(* LS Electric XG5000 project: elevator *)
(* PLC LSPLC *)
(* module base 0 slot 0: FEnet:XGL-EFMT(B) (Fast Ethernet 통신 모듈, 전기 Master) *)
(* module base 0 slot 1: 입력 모듈:XGI-D21A (DC 24V 입력, 8점 (전류소스/싱크입력)) *)
(* module base 0 slot 2: 출력 모듈:XGQ-RY1A (릴레이 출력, 8점 (2A용, 단독 COM.)) *)

(* Comments on direct variables
%IX0.1.0	1층 외부 ▲
%IX0.1.1	2층 외부  ▲
%IX0.1.2	2층 외부 ▼
%IX0.1.3	3층 외부  ▲
%IX0.1.4	3층 외부 ▼
%IX0.1.5	4층 외부  ▲
%IX0.1.6	4층 외부 ▼
%IX0.1.7	5층 외부 ▼
%IX0.3.0	내부 목적지 1F
%IX0.3.1	내부 목적지 2F
%IX0.3.2	내부 목적지 3F
%IX0.3.3	내부 목적지 4F
%IX0.3.4	내부 목적지 5F
%IX0.3.5	문 열기
%IX0.3.6	문 닫기
%IX0.3.7	비상정지
%MX80	1층 상승
%MX81	2층 상승
%MX82	3층 상승
%MX83	4층 상승
%MX89	2층 하강
%MX90	3층 하강
%MX91	4층 하강
%MX92	5층 하강
%MX96	1층
%MX97	2층
%MX98	3층
%MX99	4층
%MX100	5층
%MX160	비상정지
%MX161	문 닫힘 / 이동 가능
%MX162	문 열리는 중
%MX163	문 완전 열림
%MX164	문 딛히는 중
%MX165	상승 가능
%MX166	하강 가능
%MX167	초기화용
%MX176	1층 호출 있음
%MX177	2층 호출 있음
%MX178	3층 호출 있음
%MX179	4층 호출 있음
%MX180	5층 호출 있음
%MX181	내부 큐 있음
%MX240	외부 입력 1▲
%MX241	외부 입력 2▲
%MX242	외부 입력 2▼
%MX243	외부 입력 3▲
%MX244	외부 입력 3▼
%MX245	외부 입력 4▲
%MX246	외부 입력 4▼
%MX247	외부 입력 5▼
%MX248	내부 입력 1F
%MX249	내부 입력 2F
%MX250	내부 입력 3F
%MX251	내부 입력 4F
%MX252	내부 입력 5F
%MX253	내부입력 문열기
%MX254	내부입력 문닫기
%MX255	내부 비상정지
%MB10	상승 큐
%MB11	하강 큐
%MB12	내부 큐
%MW0	현재 층
%MW1	목표 층
%MW2	이동 방향
%MW3	상태
%MW4	TO.ET 전달용
%QX0.4.0	1층 표시등
%QX0.4.1	2층 표시등
%QX0.4.2	3층 표시등
%QX0.4.3	4층 표시등
%QX0.4.4	5층 표시등
%QX0.4.5	상승 ▲ 표시등
%QX0.4.6	하강 ▼ 표시등
%QX0.4.7	비상정지 표시등
*)

PROGRAM 리셋 (* task: 스캔 프로그램 *)
VAR
    _p1 : BOOL;
END_VAR

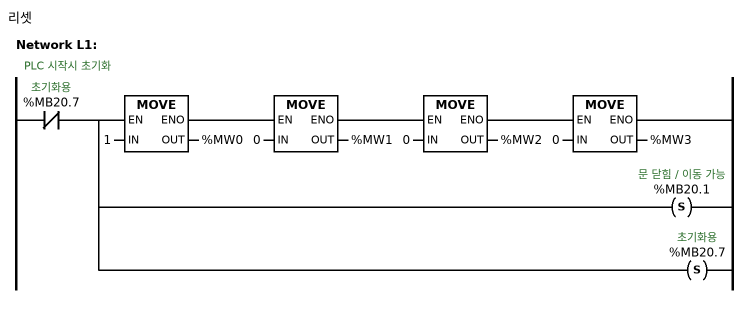
(* PLC 시작시 초기화 *)
(* Rung L1 *)
IF NOT %MB20.7 THEN
    %MW0 := 1;
    %MW1 := 0;
    %MW2 := 0;
    %MW3 := 0;
END_IF;
_p1 := NOT %MB20.7;
IF _p1 THEN
    %MB20.1 := TRUE;
    %MB20.7 := TRUE;
END_IF;
END_PROGRAM

PROGRAM 비상정지 (* task: 스캔 프로그램 *)
VAR
    _p1 : BOOL;
    _p2 : BOOL;
END_VAR

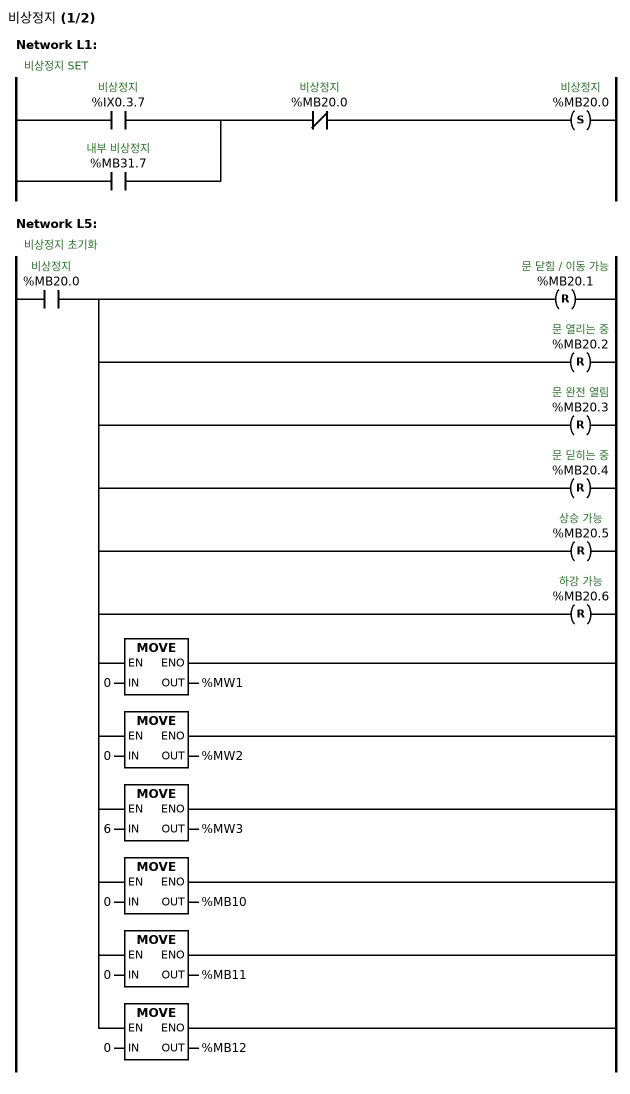
(* 비상정지 SET *)
(* Rung L1 *)
IF (%IX0.3.7 OR %MB31.7) AND NOT %MB20.0 THEN %MB20.0 := TRUE; END_IF;
(* 비상정지 초기화 *)
(* Rung L5 *)
_p1 := %MB20.0;
IF _p1 THEN
    %MB20.1 := FALSE;
    %MB20.2 := FALSE;
    %MB20.3 := FALSE;
    %MB20.4 := FALSE;
    %MB20.5 := FALSE;
    %MB20.6 := FALSE;
    %MW1 := 0;
    %MW2 := 0;
    %MW3 := 6;
    %MB10 := 0;
    %MB11 := 0;
    %MB12 := 0;
END_IF;

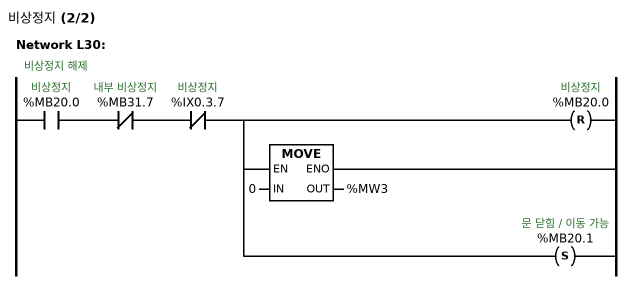
(* 비상정지 해제 *)
(* Rung L30 *)
_p2 := %MB20.0 AND NOT %MB31.7 AND NOT %IX0.3.7;
IF _p2 THEN
    %MB20.0 := FALSE;
    %MW3 := 0;
    %MB20.1 := TRUE;
END_IF;
END_PROGRAM

PROGRAM 호출큐등록 (* task: 스캔 프로그램 *)

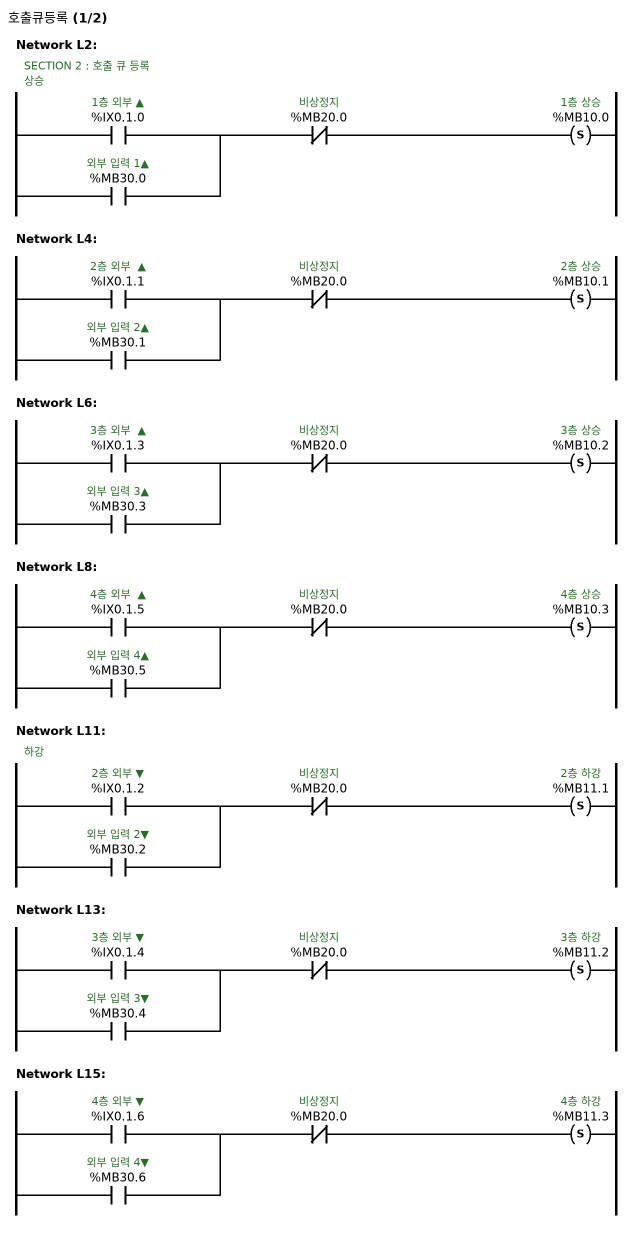
(* SECTION 2 : 호출 큐 등록 *)
(* 상승 *)
(* Rung L2 *)
IF (%IX0.1.0 OR %MB30.0) AND NOT %MB20.0 THEN %MB10.0 := TRUE; END_IF;
(* Rung L4 *)
IF (%IX0.1.1 OR %MB30.1) AND NOT %MB20.0 THEN %MB10.1 := TRUE; END_IF;
(* Rung L6 *)
IF (%IX0.1.3 OR %MB30.3) AND NOT %MB20.0 THEN %MB10.2 := TRUE; END_IF;
(* Rung L8 *)
IF (%IX0.1.5 OR %MB30.5) AND NOT %MB20.0 THEN %MB10.3 := TRUE; END_IF;
(* 하강 *)
(* Rung L11 *)
IF (%IX0.1.2 OR %MB30.2) AND NOT %MB20.0 THEN %MB11.1 := TRUE; END_IF;
(* Rung L13 *)
IF (%IX0.1.4 OR %MB30.4) AND NOT %MB20.0 THEN %MB11.2 := TRUE; END_IF;
(* Rung L15 *)
IF (%IX0.1.6 OR %MB30.6) AND NOT %MB20.0 THEN %MB11.3 := TRUE; END_IF;

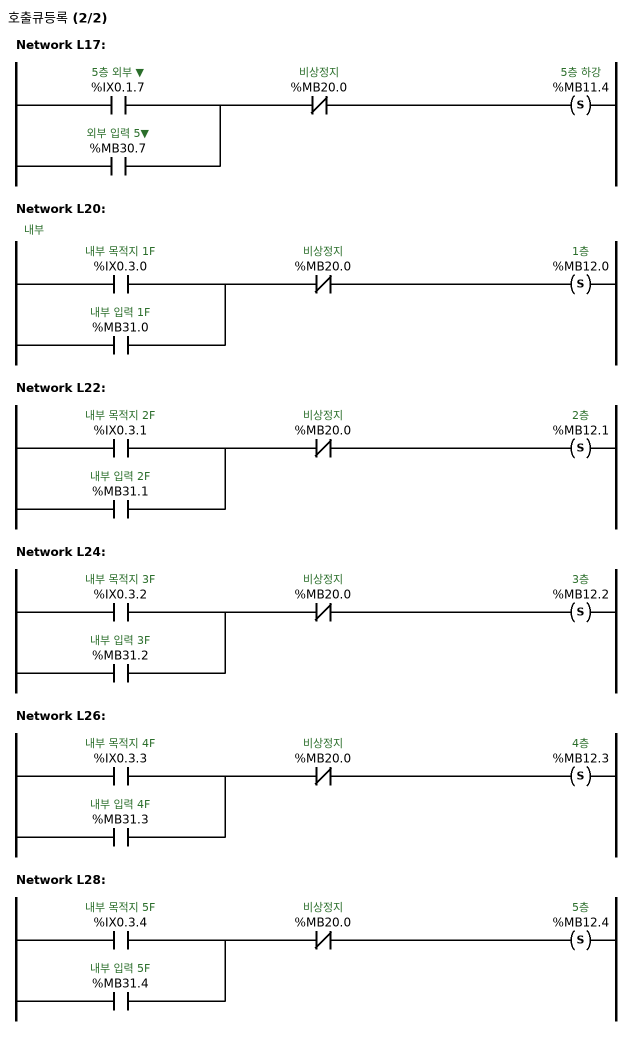
(* Rung L17 *)
IF (%IX0.1.7 OR %MB30.7) AND NOT %MB20.0 THEN %MB11.4 := TRUE; END_IF;
(* 내부 *)
(* Rung L20 *)
IF (%IX0.3.0 OR %MB31.0) AND NOT %MB20.0 THEN %MB12.0 := TRUE; END_IF;
(* Rung L22 *)
IF (%IX0.3.1 OR %MB31.1) AND NOT %MB20.0 THEN %MB12.1 := TRUE; END_IF;
(* Rung L24 *)
IF (%IX0.3.2 OR %MB31.2) AND NOT %MB20.0 THEN %MB12.2 := TRUE; END_IF;
(* Rung L26 *)
IF (%IX0.3.3 OR %MB31.3) AND NOT %MB20.0 THEN %MB12.3 := TRUE; END_IF;
(* Rung L28 *)
IF (%IX0.3.4 OR %MB31.4) AND NOT %MB20.0 THEN %MB12.4 := TRUE; END_IF;
END_PROGRAM

PROGRAM 방향판별 (* task: 스캔 프로그램 *)
VAR
    _t1 : BOOL;
    _t2 : BOOL;
    _t3 : BOOL;
    _t4 : BOOL;
    _t5 : BOOL;
    _t6 : BOOL;
    _p7 : BOOL;
    _t8 : BOOL;
    _t9 : BOOL;
    _t10 : BOOL;
    _t11 : BOOL;
    _t12 : BOOL;
    _t13 : BOOL;
    _t14 : BOOL;
    _t15 : BOOL;
    _t16 : BOOL;
    _t17 : BOOL;
    _t18 : BOOL;
    _t19 : BOOL;
    _t20 : BOOL;
    _t21 : BOOL;
    _t22 : BOOL;
    _t23 : BOOL;
    _t24 : BOOL;
    _t25 : BOOL;
END_VAR

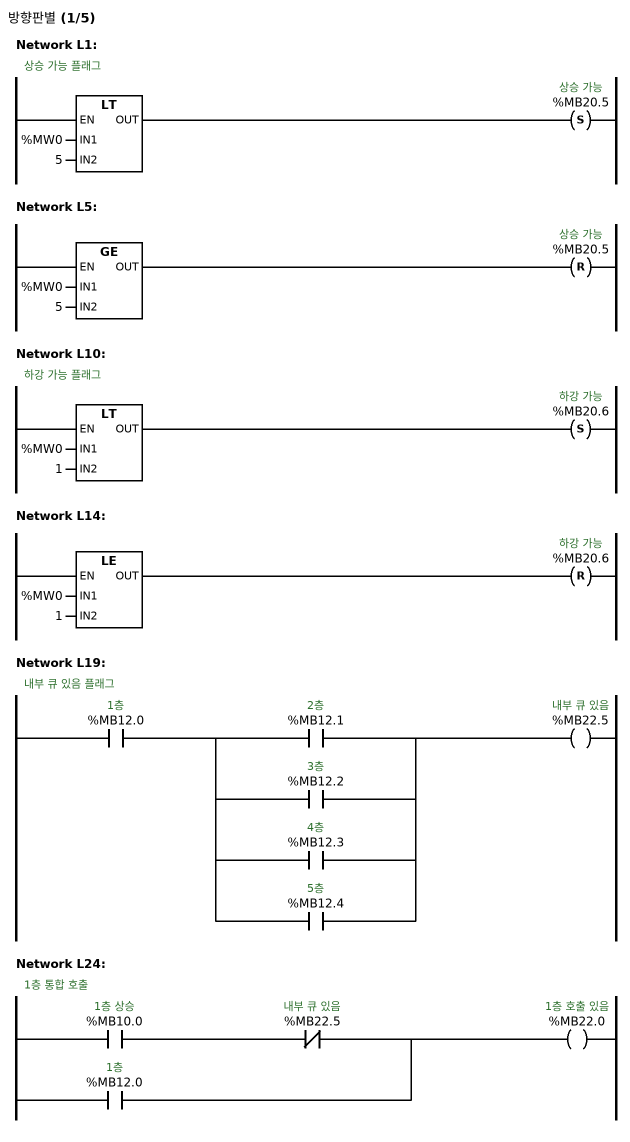
(* 상승 가능 플래그 *)
(* Rung L1 *)
IF %MW0 < 5 THEN %MB20.5 := TRUE; END_IF;
(* Rung L5 *)
IF %MW0 >= 5 THEN %MB20.5 := FALSE; END_IF;
(* 하강 가능 플래그 *)
(* Rung L10 *)
IF %MW0 < 1 THEN %MB20.6 := TRUE; END_IF;
(* Rung L14 *)
IF %MW0 <= 1 THEN %MB20.6 := FALSE; END_IF;
(* 내부 큐 있음 플래그 *)
(* Rung L19 *)
%MB22.5 := %MB12.0 AND (%MB12.1 OR %MB12.2 OR %MB12.3 OR %MB12.4);
(* 1층 통합 호출 *)
(* Rung L24 *)
%MB22.0 := (%MB10.0 AND NOT %MB22.5) OR %MB12.0;

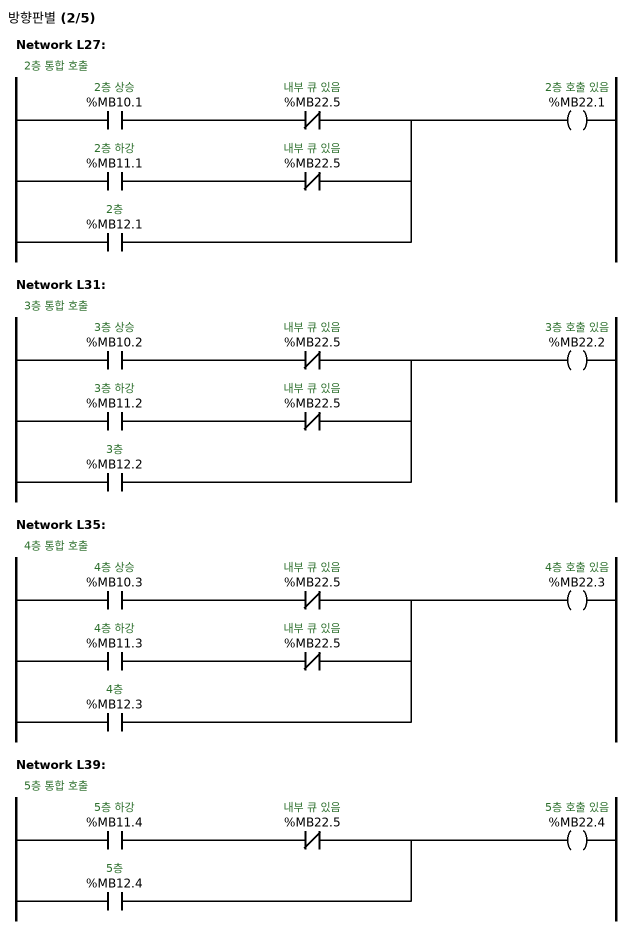
(* 2층 통합 호출 *)
(* Rung L27 *)
%MB22.1 := (%MB10.1 AND NOT %MB22.5) OR (%MB11.1 AND NOT %MB22.5) OR %MB12.1;
(* 3층 통합 호출 *)
(* Rung L31 *)
%MB22.2 := (%MB10.2 AND NOT %MB22.5) OR (%MB11.2 AND NOT %MB22.5) OR %MB12.2;
(* 4층 통합 호출 *)
(* Rung L35 *)
%MB22.3 := (%MB10.3 AND NOT %MB22.5) OR (%MB11.3 AND NOT %MB22.5) OR %MB12.3;
(* 5층 통합 호출 *)
(* Rung L39 *)
%MB22.4 := (%MB11.4 AND NOT %MB22.5) OR %MB12.4;

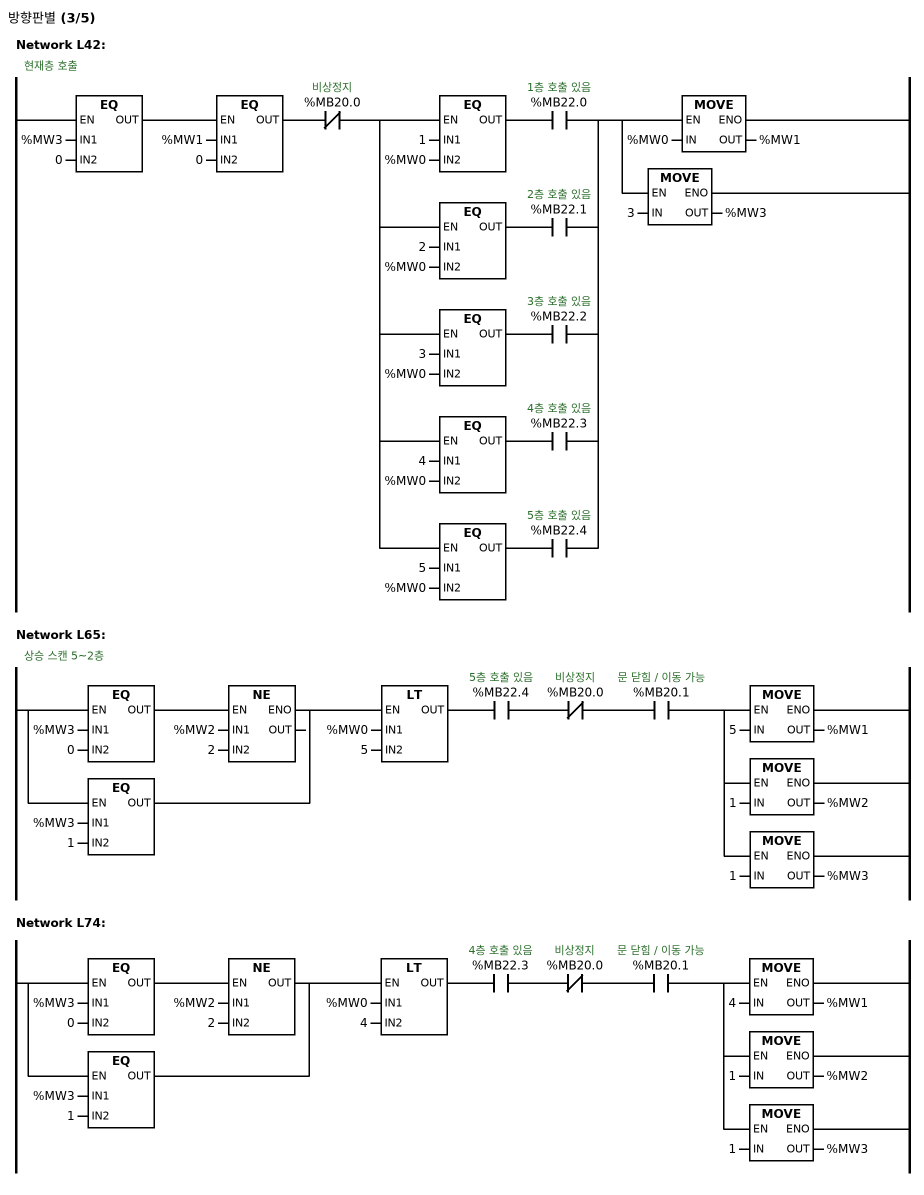
(* 현재층 호출 *)
(* Rung L42 *)
IF %MW3 = 0 THEN _t1 := %MW1 = 0; END_IF;
IF _t1 AND NOT %MB20.0 THEN
    _t2 := 1 = %MW0;
    _t3 := 2 = %MW0;
    _t4 := 3 = %MW0;
    _t5 := 4 = %MW0;
    _t6 := 5 = %MW0;
END_IF;
_p7 := (_t2 AND %MB22.0) OR (_t3 AND %MB22.1) OR (_t4 AND %MB22.2) OR (_t5 AND %MB22.3) OR (_t6 AND %MB22.4);
IF _p7 THEN
    %MW1 := %MW0;
    %MW3 := 3;
END_IF;
(* 상승 스캔 5~2층 *)
(* Rung L65 *)
IF %MW3 = 0 THEN _t8 := %MW2 <> 2; END_IF;
IF (%MW3 = 0) OR (%MW3 = 1) THEN _t9 := %MW0 < 5; END_IF;
IF _t9 AND %MB22.4 AND NOT %MB20.0 AND %MB20.1 THEN
    %MW1 := 5;
    %MW2 := 1;
    %MW3 := 1;
END_IF;
(* Rung L74 *)
IF %MW3 = 0 THEN _t10 := %MW2 <> 2; END_IF;
IF _t10 OR (%MW3 = 1) THEN _t11 := %MW0 < 4; END_IF;
IF _t11 AND %MB22.3 AND NOT %MB20.0 AND %MB20.1 THEN
    %MW1 := 4;
    %MW2 := 1;
    %MW3 := 1;
END_IF;

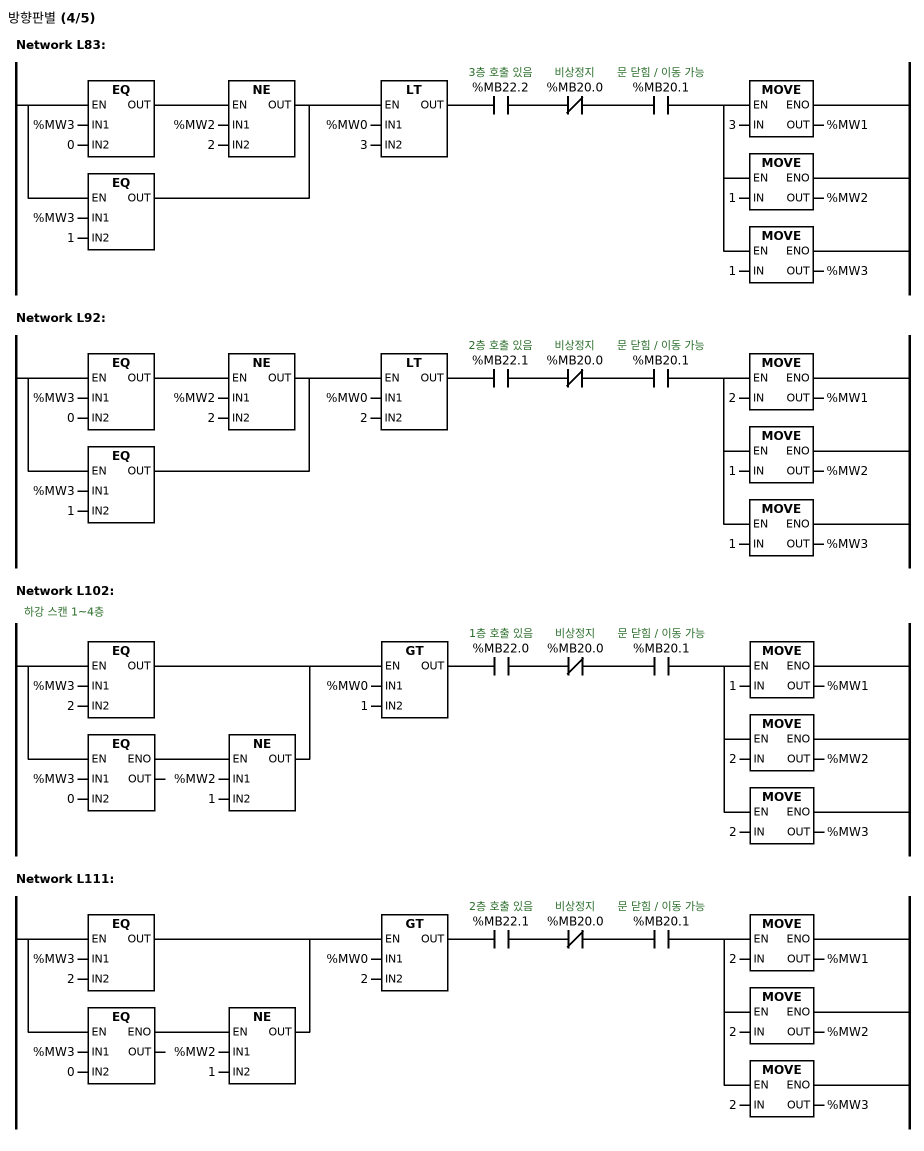
(* Rung L83 *)
IF %MW3 = 0 THEN _t12 := %MW2 <> 2; END_IF;
IF _t12 OR (%MW3 = 1) THEN _t13 := %MW0 < 3; END_IF;
IF _t13 AND %MB22.2 AND NOT %MB20.0 AND %MB20.1 THEN
    %MW1 := 3;
    %MW2 := 1;
    %MW3 := 1;
END_IF;
(* Rung L92 *)
IF %MW3 = 0 THEN _t14 := %MW2 <> 2; END_IF;
IF _t14 OR (%MW3 = 1) THEN _t15 := %MW0 < 2; END_IF;
IF _t15 AND %MB22.1 AND NOT %MB20.0 AND %MB20.1 THEN
    %MW1 := 2;
    %MW2 := 1;
    %MW3 := 1;
END_IF;
(* 하강 스캔 1~4층 *)
(* Rung L102 *)
_t16 := %MW3 = 0;
IF (%MW3 = 2) OR (%MW2 <> 1) THEN _t17 := %MW0 > 1; END_IF;
IF _t17 AND %MB22.0 AND NOT %MB20.0 AND %MB20.1 THEN
    %MW1 := 1;
    %MW2 := 2;
    %MW3 := 2;
END_IF;
(* Rung L111 *)
_t18 := %MW3 = 0;
IF (%MW3 = 2) OR (%MW2 <> 1) THEN _t19 := %MW0 > 2; END_IF;
IF _t19 AND %MB22.1 AND NOT %MB20.0 AND %MB20.1 THEN
    %MW1 := 2;
    %MW2 := 2;
    %MW3 := 2;
END_IF;

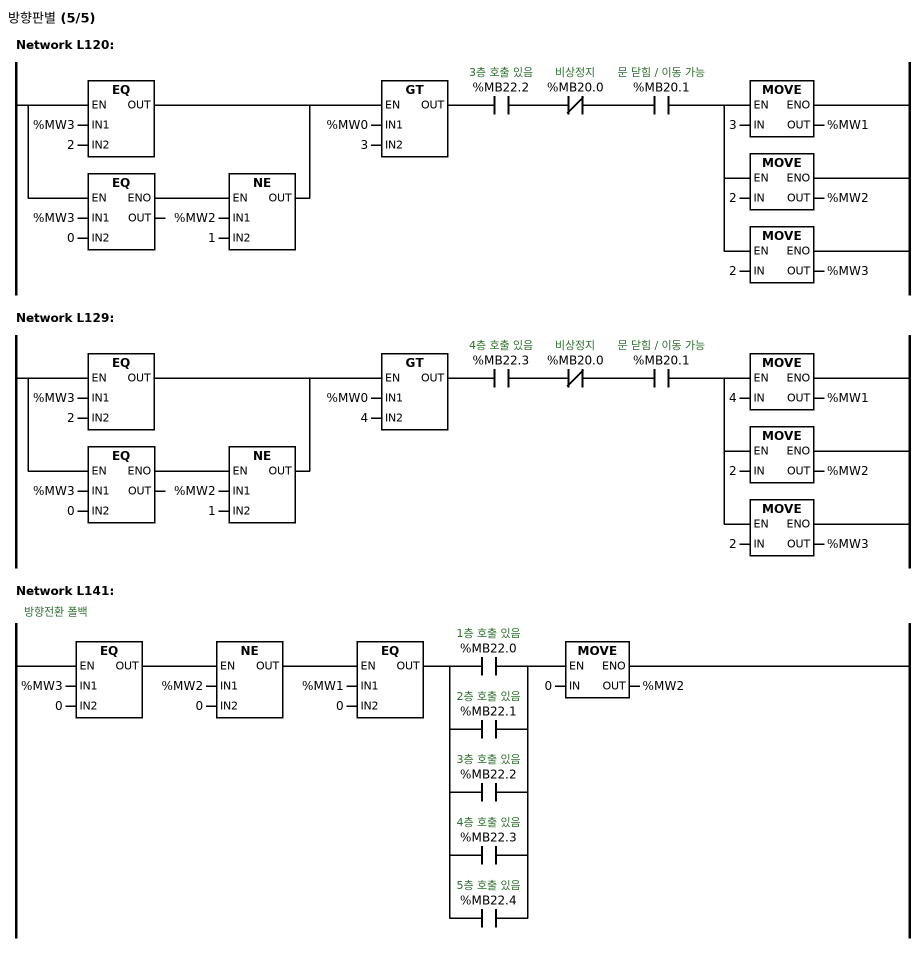
(* Rung L120 *)
_t20 := %MW3 = 0;
IF (%MW3 = 2) OR (%MW2 <> 1) THEN _t21 := %MW0 > 3; END_IF;
IF _t21 AND %MB22.2 AND NOT %MB20.0 AND %MB20.1 THEN
    %MW1 := 3;
    %MW2 := 2;
    %MW3 := 2;
END_IF;
(* Rung L129 *)
_t22 := %MW3 = 0;
IF (%MW3 = 2) OR (%MW2 <> 1) THEN _t23 := %MW0 > 4; END_IF;
IF _t23 AND %MB22.3 AND NOT %MB20.0 AND %MB20.1 THEN
    %MW1 := 4;
    %MW2 := 2;
    %MW3 := 2;
END_IF;
(* 방향전환 폴백 *)
(* Rung L141 *)
IF %MW3 = 0 THEN _t24 := %MW2 <> 0; END_IF;
IF _t24 THEN _t25 := %MW1 = 0; END_IF;
IF _t25 AND (%MB22.0 OR %MB22.1 OR %MB22.2 OR %MB22.3 OR %MB22.4) THEN %MW2 := 0; END_IF;
END_PROGRAM

PROGRAM 이동제어 (* task: 스캔 프로그램 *)
VAR
    T4 : TON;
    T5 : TON;
    T6 : TON;
END_VAR
VAR
    _t1 : BOOL;
    _t2 : BOOL;
    _t3 : BOOL;
    _t4 : BOOL;
    _t5 : BOOL;
END_VAR

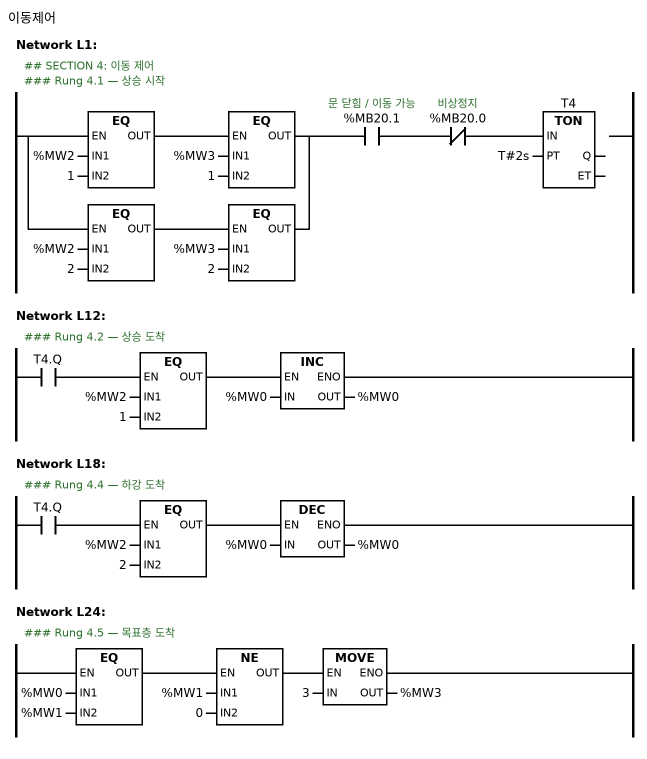
(* ## SECTION 4: 이동 제어 / ### Rung 4.1 — 상승 시작 *)
(* Rung L1 *)
IF %MW2 = 1 THEN _t1 := %MW3 = 1; END_IF;
IF %MW2 = 2 THEN _t2 := %MW3 = 2; END_IF;
T4(IN := (_t1 OR _t2) AND %MB20.1 AND NOT %MB20.0, PT := T#2s);
(* ### Rung 4.2 — 상승 도착 *)
(* Rung L12 *)
IF T4.Q THEN _t3 := %MW2 = 1; END_IF;
IF _t3 THEN %MW0 := INC(%MW0); END_IF;
(* ### Rung 4.4 — 하강 도착 *)
(* Rung L18 *)
IF T4.Q THEN _t4 := %MW2 = 2; END_IF;
IF _t4 THEN %MW0 := DEC(%MW0); END_IF;
(* ### Rung 4.5 — 목표층 도착 *)
(* Rung L24 *)
IF %MW0 = %MW1 THEN _t5 := %MW1 <> 0; END_IF;
IF _t5 THEN %MW3 := 3; END_IF;
END_PROGRAM

PROGRAM 도착큐클리어 (* task: 스캔 프로그램 *)
VAR
    _t1 : BOOL;
    _t2 : BOOL;
    _t3 : BOOL;
    _t4 : BOOL;
    _t5 : BOOL;
END_VAR

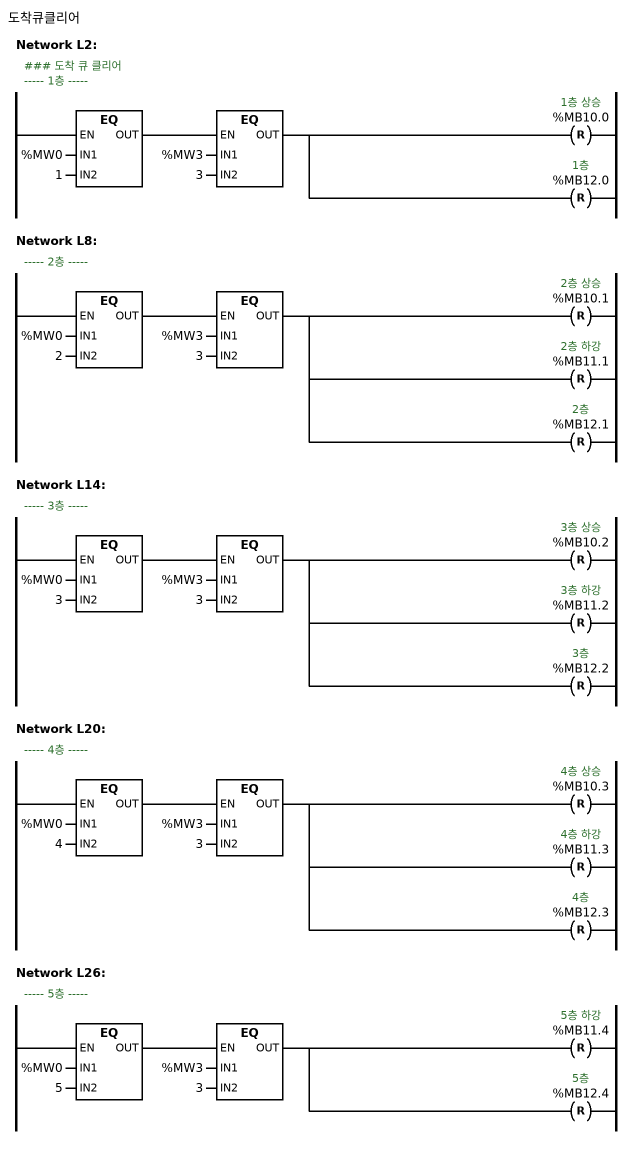
(* ### 도착 큐 클리어 *)
(* ----- 1층 ----- *)
(* Rung L2 *)
IF %MW0 = 1 THEN _t1 := %MW3 = 3; END_IF;
IF _t1 THEN
    %MB10.0 := FALSE;
    %MB12.0 := FALSE;
END_IF;
(* ----- 2층 ----- *)
(* Rung L8 *)
IF %MW0 = 2 THEN _t2 := %MW3 = 3; END_IF;
IF _t2 THEN
    %MB10.1 := FALSE;
    %MB11.1 := FALSE;
    %MB12.1 := FALSE;
END_IF;
(* ----- 3층 ----- *)
(* Rung L14 *)
IF %MW0 = 3 THEN _t3 := %MW3 = 3; END_IF;
IF _t3 THEN
    %MB10.2 := FALSE;
    %MB11.2 := FALSE;
    %MB12.2 := FALSE;
END_IF;
(* ----- 4층 ----- *)
(* Rung L20 *)
IF %MW0 = 4 THEN _t4 := %MW3 = 3; END_IF;
IF _t4 THEN
    %MB10.3 := FALSE;
    %MB11.3 := FALSE;
    %MB12.3 := FALSE;
END_IF;
(* ----- 5층 ----- *)
(* Rung L26 *)
IF %MW0 = 5 THEN _t5 := %MW3 = 3; END_IF;
IF _t5 THEN
    %MB11.4 := FALSE;
    %MB12.4 := FALSE;
END_IF;
END_PROGRAM

PROGRAM 문제어 (* task: 스캔 프로그램 *)
VAR
    T0 : TON;
    T1 : TON;
    T2 : TON;
END_VAR
VAR
    _p1 : BOOL;
    _p2 : BOOL;
    _p3 : BOOL;
    _t4 : BOOL;
    _p5 : BOOL;
END_VAR

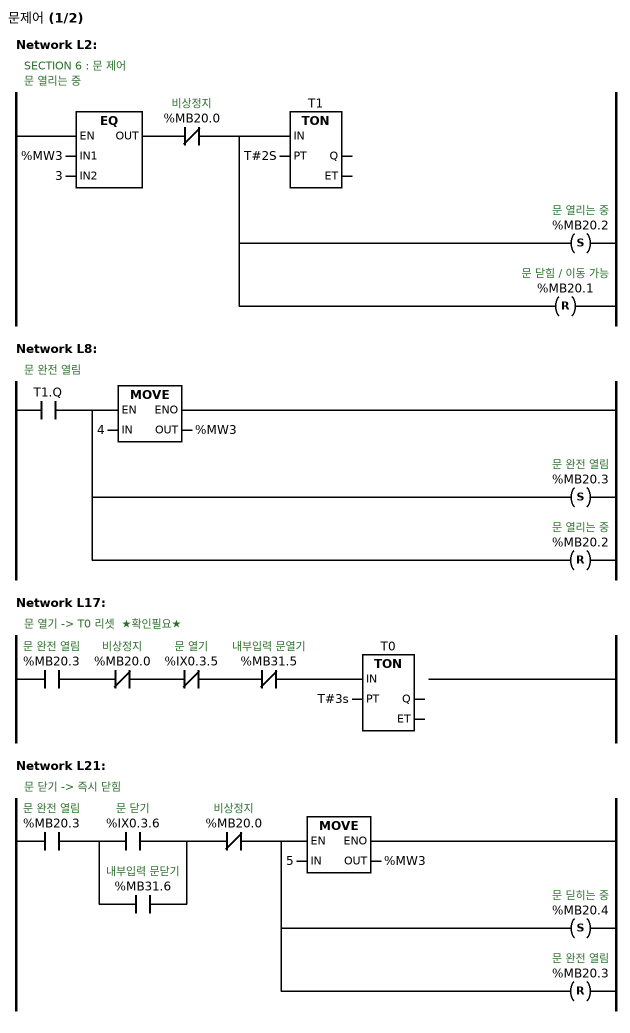
(* SECTION 6 : 문 제어 *)
(* 문 열리는 중 *)
(* Rung L2 *)
T1(IN := (%MW3 = 3) AND NOT %MB20.0, PT := T#2S);
_p1 := (%MW3 = 3) AND NOT %MB20.0;
IF _p1 THEN
    %MB20.2 := TRUE;
    %MB20.1 := FALSE;
END_IF;
(* 문 완전 열림 *)
(* Rung L8 *)
IF T1.Q THEN
    %MW3 := 4;
    %MB20.3 := TRUE;
    %MB20.2 := FALSE;
END_IF;
(* 문 열기 -> T0 리셋  ★확인필요★ *)
(* Rung L17 *)
T0(IN := %MB20.3 AND NOT %MB20.0 AND NOT %IX0.3.5 AND NOT %MB31.5, PT := T#3s);
(* 문 닫기 -> 즉시 닫힘 *)
(* Rung L21 *)
_p2 := %MB20.3 AND (%IX0.3.6 OR %MB31.6) AND NOT %MB20.0;
IF _p2 THEN
    %MW3 := 5;
    %MB20.4 := TRUE;
    %MB20.3 := FALSE;
END_IF;

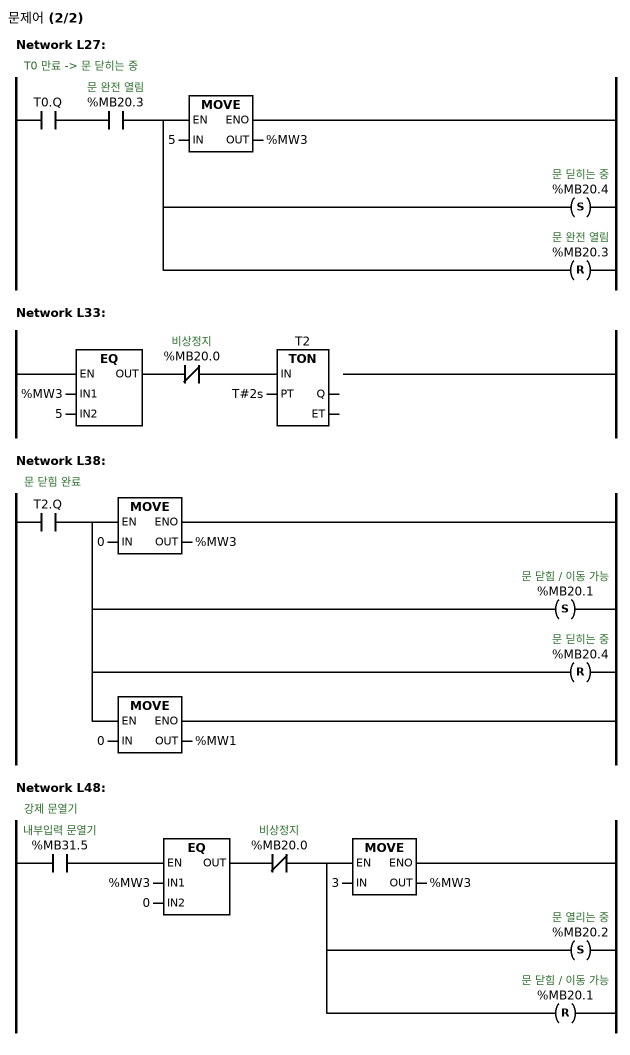
(* T0 만료 -> 문 닫히는 중 *)
(* Rung L27 *)
IF T0.Q AND %MB20.3 THEN %MW3 := 5; END_IF;
_p3 := T0.Q AND %MB20.3;
IF _p3 THEN
    %MB20.4 := TRUE;
    %MB20.3 := FALSE;
END_IF;
(* Rung L33 *)
T2(IN := (%MW3 = 5) AND NOT %MB20.0, PT := T#2s);
(* 문 닫힘 완료 *)
(* Rung L38 *)
IF T2.Q THEN
    %MW3 := 0;
    %MB20.1 := TRUE;
    %MB20.4 := FALSE;
    %MW1 := 0;
END_IF;
(* 강제 문열기 *)
(* Rung L48 *)
IF %MB31.5 THEN _t4 := %MW3 = 0; END_IF;
IF _t4 AND NOT %MB20.0 THEN %MW3 := 3; END_IF;
_p5 := _t4 AND NOT %MB20.0;
IF _p5 THEN
    %MB20.2 := TRUE;
    %MB20.1 := FALSE;
END_IF;
END_PROGRAM

PROGRAM 인터락 (* task: 스캔 프로그램 *)

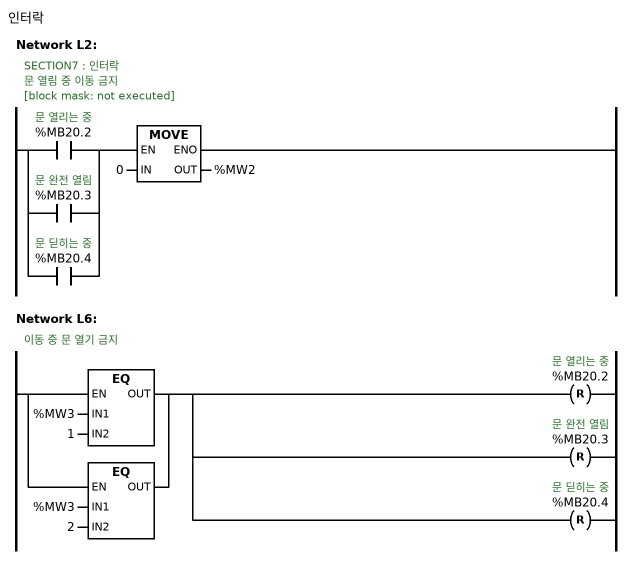
(* SECTION7 : 인터락 *)
(* 문 열림 중 이동 금지 *)
(* Rung L2 is block-masked: not executed *)
// IF %MB20.2 OR %MB20.3 OR %MB20.4 THEN %MW2 := 0; END_IF;
(* 이동 중 문 열기 금지 *)
(* Rung L6 *)
IF (%MW3 = 1) OR (%MW3 = 2) THEN
    %MB20.2 := FALSE;
    %MB20.3 := FALSE;
    %MB20.4 := FALSE;
END_IF;
END_PROGRAM

PROGRAM 출력표시등 (* task: 스캔 프로그램 *)

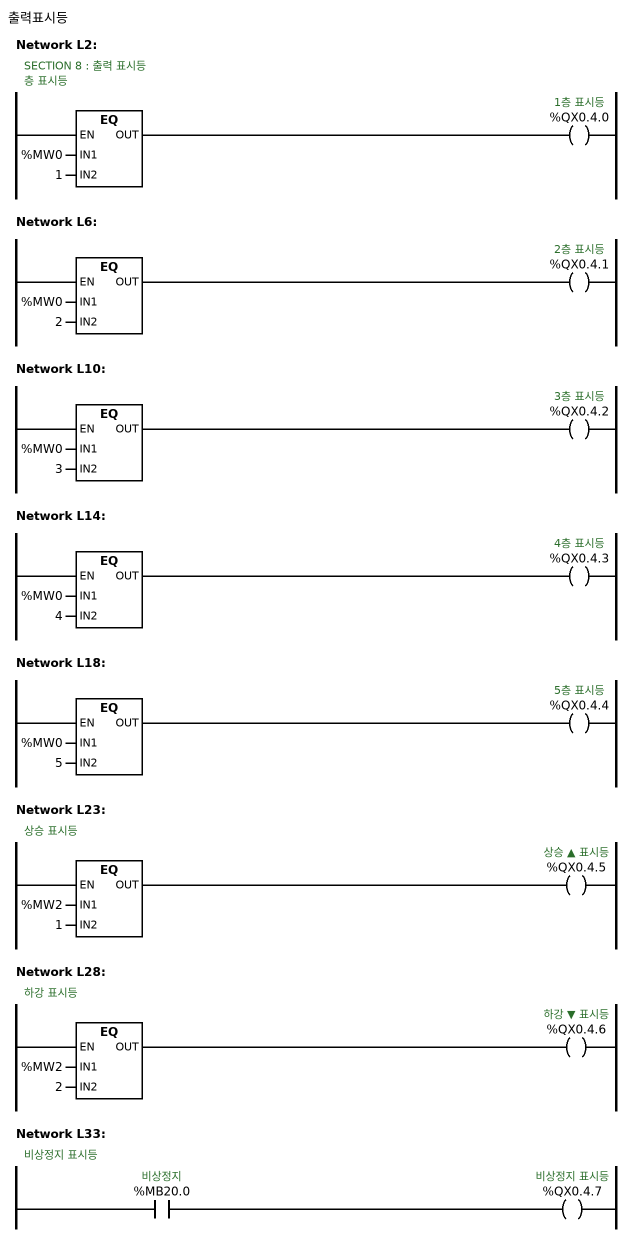
(* SECTION 8 : 출력 표시등 *)
(* 층 표시등 *)
(* Rung L2 *)
%QX0.4.0 := %MW0 = 1;
(* Rung L6 *)
%QX0.4.1 := %MW0 = 2;
(* Rung L10 *)
%QX0.4.2 := %MW0 = 3;
(* Rung L14 *)
%QX0.4.3 := %MW0 = 4;
(* Rung L18 *)
%QX0.4.4 := %MW0 = 5;
(* 상승 표시등 *)
(* Rung L23 *)
%QX0.4.5 := %MW2 = 1;
(* 하강 표시등 *)
(* Rung L28 *)
%QX0.4.6 := %MW2 = 2;
(* 비상정지 표시등 *)
(* Rung L33 *)
%QX0.4.7 := %MB20.0;
END_PROGRAM